{attribute addProperty BoxType "EL5021-0000-0016"}
{attribute addProperty Id "Latch_C_validBIT10.1251Set_counter_doneBIT10.1253Frequency_errorBIT10.1254Amplitude_errorBIT10.1255Status_of_input_CBIT10.12511Sync_errorBIT10.12532TxPDO_StateBIT10.1257TxPDO_ToggleBIT10.1259"}
{attribute addProperty CRC "1342784561"}
{attribute addProperty SizeInBites "16"}
{attribute addProperty SizeInBytes "2"}
TYPE Status_50094431 :
STRUCT
	{attribute addProperty Name "Latch_C_valid"}
	Latch_C_valid : BIT;
	{attribute 'hide'}
	reserve_1 : BIT;
	{attribute addProperty Name "Set_counter_done"}
	Set_counter_done : BIT;
	{attribute addProperty Name "Frequency_error"}
	Frequency_error : BIT;
	{attribute addProperty Name "Amplitude_error"}
	Amplitude_error : BIT;
	{attribute 'hide'}
	reserve_2_BIT_0 : BIT;
	{attribute 'hide'}
	reserve_2_BIT_1 : BIT;
	{attribute 'hide'}
	reserve_2_BIT_2 : BIT;
	{attribute 'hide'}
	reserve_2_BIT_3 : BIT;
	{attribute 'hide'}
	reserve_2_BIT_4 : BIT;
	{attribute addProperty Name "Status_of_input_C"}
	Status_of_input_C : BIT;
	{attribute 'hide'}
	reserve_3_BIT_0 : BIT;
	{attribute 'hide'}
	reserve_3_BIT_1 : BIT;
	{attribute addProperty Name "Sync_error"}
	Sync_error : BIT;
	{attribute addProperty Name "TxPDO_State"}
	TxPDO_State : BIT;
	{attribute addProperty Name "TxPDO_Toggle"}
	TxPDO_Toggle : BIT;
END_STRUCT
END_TYPE

(* stored: Version 1.2.0.0, ProductVersion 3.1.4024.9
   DUT Status_50094431: Id {097f3bc2-f908-4ee9-bf1f-222c17c463ad} *)
